// TIA Portal V17 export
// export: Created 2024-10-17T14:16:19.5103777Z, ExportSetting WithDefaults, DisplayName Totally Integrated Automation Portal, DisplayVersion V17 Update 4, DisplayName TIA Portal Openness, DisplayVersion V17 Update 4, DisplayName TIA Portal Version Control Interface, DisplayVersion V17, DisplayName SINAMICS Startdrive Advanced, DisplayVersion V17 Update2, DisplayName SINAMICS Startdrive G130, G150, S120, S150, SINAMICS MV, S210, DisplayVersion V17 Update2, DisplayName SINAMICS Startdrive G110M, G120, G120C, G120D, G120P, G115D, DisplayVersion V17 Update2, DisplayName STEP 7 Professional, DisplayVersion V17 Update 4, DisplayName STEP 7 Safety, DisplayVersion V17, DisplayName WinCC Advanced / Unified PC, DisplayVersion V17 Update 4
DATA_BLOCK "InstLPMLV2022_UnitModeStateManagerBool"   // DB30111
{ DB_Accessible_From_OPC_UA := 'FALSE' }
AUTHOR : APC_ERLF
FAMILY : OMAC
VERSION : 1.0
// stored: AutoNumber true, DBAccessibleFromOPCUA false, InstanceOfName LPMLV2022_UnitModeStateManagerBool, InstanceOfType FB
"LPMLV2022_UnitModeStateManagerBool"
   // VAR_INPUT
   //    ProductionModeRequest : Bool;
   //    MaintenanceModeRequest : Bool;
   //    ManualModeRequest : Bool;
   //    UserMode01Request : Bool;
   //    UserMode02Request : Bool;
   //    UserMode03Request : Bool;
   //    UserMode04Request : Bool;
   //    UserMode05Request : Bool;
   //    ResetCmdRequest : Bool;
   //    StartCmdRequest : Bool;
   //    StopCmdRequest : Bool;
   //    HoldCmdRequest : Bool;
   //    UnholdCmdRequest : Bool;
   //    SuspendCmdRequest : Bool;
   //    UnsuspendCmdRequest : Bool;
   //    AbortCmdRequest : Bool;
   //    ClearCmdRequest : Bool;
   //    CompleteCmdRequest : Bool;
   //    SC : Bool;
   //    configuration : "LPMLV2022_typeConfiguration";
   // END_VAR
   // VAR_OUTPUT
   //    UnitModeCurrent { ExternalWritable := 'False'} : DInt;
   //    StateCurrent { ExternalWritable := 'False'} : DInt;
   //    ProductionModeActive { ExternalWritable := 'False'} : Bool;
   //    MaintenanceModeActive { ExternalWritable := 'False'} : Bool;
   //    ManualModeActive { ExternalWritable := 'False'} : Bool;
   //    UserMode01Active { ExternalWritable := 'False'} : Bool;
   //    UserMode02Active { ExternalWritable := 'False'} : Bool;
   //    UserMode03Active { ExternalWritable := 'False'} : Bool;
   //    UserMode04Active { ExternalWritable := 'False'} : Bool;
   //    UserMode05Active { ExternalWritable := 'False'} : Bool;
   //    ClearingStateActive { ExternalWritable := 'False'} : Bool;
   //    StoppedStateActive { ExternalWritable := 'False'} : Bool;
   //    StartingStateActive { ExternalWritable := 'False'} : Bool;
   //    IdleStateActive { ExternalWritable := 'False'} : Bool;
   //    SuspendedStateActive { ExternalWritable := 'False'} : Bool;
   //    ExecuteStateActive { ExternalWritable := 'False'} : Bool;
   //    StoppingStateActive { ExternalWritable := 'False'} : Bool;
   //    AbortingStateActive { ExternalWritable := 'False'} : Bool;
   //    AbortedStateActive { ExternalWritable := 'False'} : Bool;
   //    HoldingStateActive { ExternalWritable := 'False'} : Bool;
   //    HeldStateActive { ExternalWritable := 'False'} : Bool;
   //    UnholdingStateActive { ExternalWritable := 'False'} : Bool;
   //    SuspendingStateActive { ExternalWritable := 'False'} : Bool;
   //    UnsuspendingStateActive { ExternalWritable := 'False'} : Bool;
   //    ResettingStateActive { ExternalWritable := 'False'} : Bool;
   //    CompletingStateActive { ExternalWritable := 'False'} : Bool;
   //    CompletedStateActive { ExternalWritable := 'False'} : Bool;
   //    unitModeChangeNotAllowed { ExternalWritable := 'False'} : Bool;
   //    cntrlCmdNotAllowed { ExternalWritable := 'False'} : Bool;
   // END_VAR
   // VAR
   //    instUnitModeStateManager { ExternalWritable := 'False'} : "LPMLV2022_UnitModeStateManager";
   //    statFirstCycle { ExternalAccessible := 'False'; ExternalVisible := 'False'; ExternalWritable := 'False'} : Bool;
   //    statUnitModeCurrentInternalOld { ExternalAccessible := 'False'; ExternalVisible := 'False'; ExternalWritable := 'False'} : DInt;
   //    statStateInternalOld { ExternalAccessible := 'False'; ExternalVisible := 'False'; ExternalWritable := 'False'} : DInt;
   //    statBooleanInterfaceModeOld { ExternalAccessible := 'False'; ExternalVisible := 'False'; ExternalWritable := 'False'} : DWord;
   //    statBooleanInterfaceCmdOld { ExternalAccessible := 'False'; ExternalVisible := 'False'; ExternalWritable := 'False'} : Word;
   // END_VAR
BEGIN
END_DATA_BLOCK
